RoboDK station: New Station (1).rdk

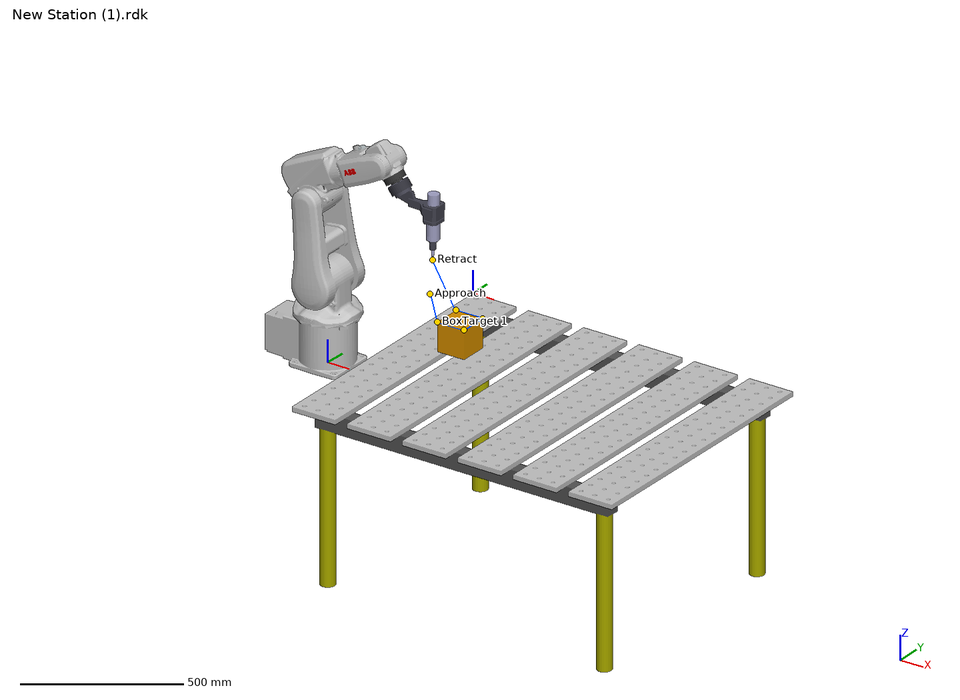
[picture v0: the station drawn from its stored meshes, robots at their saved joint values, targets as dots, program paths as lines]
Station New Station (1) (saved by RoboDK 5.2.3). Poses are relative to the parent item; angles as X-Y-Z fixed-axis rotations.
  - frame ABB IRB 120-3/0.6 Base at (0, 0, 0) mm
    - robot ABB IRB 120-3/0.6: 6 axes, payload 3 kg, reach 580 mm, repeatability 0.01 mm, weight 25 kg
        modified DH rows (alpha deg, a mm, theta deg, d mm): 0, 0, 0, 290; -90, 0, -90, 0; 0, 270, 0, 0; -90, 70, 0, 302; 90, 0, 0, 0; -90, 0, 180, 72
        joint limits [-165, -110, -90, -160, -120, -400] to [165, 110, 70, 160, 120, 400]; home [0, 0, 0, 0, 0, 0]; saved at [-0.259, -6.594, -17.186, 0.16, 76.75, -0.243]
      - tool Spintech Spindle, TCP at (32, 0, 260) mm, rotated rx 0 ry 39 rz 0 deg, size 157.3 x 72 x 259.9 mm
  - object Table 1200x1000mm (Welding) at (800, 0, 100) mm, size 1193.8 x 965.2 x 609.6 mm, geometry from Table-1200x1000mm-Welding.sld
  - frame Worktable at (203.1, 482.6, 100) mm, rotated rx 0 ry 0 rz 0.28 deg
    - object Cube 100mm at (200, -480, 50) mm, size 100 x 100 x 100 mm, geometry from Cube-100mm.sld
    - target Approach (Cartesian target) at (177.65, -484.46, 240.96) mm, rotated rx -180 ry -1.97 rz 179.72 deg; joints [-0.269, -19.59, 17.512, 0.198, 55.049, -0.328] of ABB IRB 120-3/0.6
    - target Retract (Cartesian target) at (186.05, -484.5, 359.73) mm, rotated rx -180 ry -1.97 rz 179.72 deg; joints [-0.259, -6.594, -17.186, 0.16, 76.75, -0.243] of ABB IRB 120-3/0.6
    - target BoxTarget 1 (Cartesian target) at (200, -480, 150) mm, rotated rx 180 ry 0 rz 179.72 deg; joints [0.928, -19.049, 35.254, -1.023, 34.803, 1.562] of ABB IRB 120-3/0.6
    - target BoxTarget 2 (Cartesian target) at (300, -480, 150) mm, rotated rx 180 ry 0 rz 179.72 deg; joints [0.727, 2.762, 16.126, -0.86, 32.117, 1.294] of ABB IRB 120-3/0.6
    - target BoxTarget 3 (Cartesian target) at (300, -380, 150) mm, rotated rx -180 ry 0 rz 179.72 deg; joints [17.969, 6.129, 12.531, -19.616, 35.333, 30.359] of ABB IRB 120-3/0.6
    - target BoxTarget 4 (Cartesian target) at (200, -380, 150) mm, rotated rx 180 ry 0 rz 179.72 deg; joints [25.123, -13.954, 31.422, -25.105, 39.033, 40.022] of ABB IRB 120-3/0.6
  - program Prog1 (6 instructions, listed below)
  - program MainProgram (1 instructions, listed below)
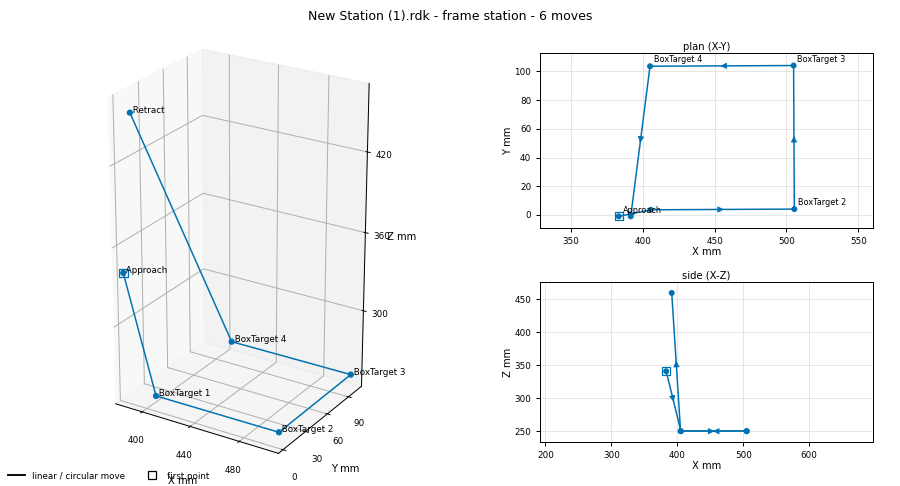
[picture p0: tool path of New Station (1).rdk in frame station, 6 of 6 moves have a stored position in this frame; points joined in program order, loops and branches not executed]

--- program Prog1 (robot ABB IRB 120-3/0.6) ---
  MoveJ (Approach)
  MoveL (BoxTarget 1)
  MoveL (BoxTarget 2)
  MoveL (BoxTarget 3)
  MoveL (BoxTarget 4)
  MoveL (Retract)

--- program MainProgram (robot ABB IRB 120-3/0.6) ---
  Call Prog1
